// TIA Portal V17 export
// export: Created 2022-07-28T18:03:21.6529657Z, ExportSetting None, DisplayName Totally Integrated Automation Portal, DisplayVersion V17, DisplayName TIA Portal Openness, DisplayVersion V17, DisplayName TIA Portal Teamcenter Gateway, DisplayVersion V17, DisplayName TIA Portal Version Control Interface, DisplayVersion V17, DisplayName TIA Portal Test Suite Advanced, DisplayVersion V17, DisplayName SINAMICS Startdrive Advanced, DisplayVersion V17, DisplayName SINAMICS DCC, DisplayVersion V17, DisplayName SINAMICS Startdrive G130, G150, S120, S150, SINAMICS MV, S210, DisplayVersion V17, DisplayName SINAMICS Startdrive G110M, G120, G120C, G120D, G120P, G115D, DisplayVersion V17, DisplayName STEP 7 Professional, DisplayVersion V17, DisplayName SIMATIC Energy Suite, DisplayVersion V17, DisplayName STEP 7 CFC, DisplayVersion V17, DisplayName STEP 7 Safety, DisplayVersion V17, DisplayName WinCC Advanced / Unified PC, DisplayVersion V17, DisplayName SIMATIC Visualization Architect, DisplayVersion V17
TYPE "_SlideGate_Cond_StateBits"
   STRUCT
      Error { ExternalAccessible := 'False'; ExternalVisible := 'False'; ExternalWritable := 'False'} : Bool;   // x0 - 1 = [1-level alarm] -General alarm- Активна Загальна аварія(об'єднує усі аварії) / General alarm - Overall error
      Warning { ExternalAccessible := 'False'; ExternalVisible := 'False'; ExternalWritable := 'False'} : Bool;   // x1 - 1 = [2-level alarm] - Warning - Активне попередження (об'єднує усі попередження)
      Maintenance { ExternalAccessible := 'False'; ExternalVisible := 'False'; ExternalWritable := 'False'} : Bool;   // x2 - 1 = [3-level ] - Maintenance - Обслуговування - Спрацювали таймери/лічильники обслуговування
      Interlocked { ExternalAccessible := 'False'; ExternalVisible := 'False'; ExternalWritable := 'False'} : Bool;   // x3 - 1 = [Interlock] - Interloked - Заблоковано
      Ready { ExternalAccessible := 'False'; ExternalVisible := 'False'; ExternalWritable := 'False'} : Bool;   // x4 - 1 = Готовий - ...........
      Stoped { ExternalAccessible := 'False'; ExternalVisible := 'False'; ExternalWritable := 'False'} : Bool;   // x5 - 1 = Зупинений
      Run { ExternalAccessible := 'False'; ExternalVisible := 'False'; ExternalWritable := 'False'} : Bool;   // x6 - 1 = Запущено / напрямок руху Forward або Revers / Відкривається або Закривається
      RunOpen { ExternalAccessible := 'False'; ExternalVisible := 'False'; ExternalWritable := 'False'} : Bool;   // x7 - 1 = Запущено / напрямок руху Forward / Відкривається
      RunClose { ExternalAccessible := 'False'; ExternalVisible := 'False'; ExternalWritable := 'False'} : Bool;   // x8 - 1 = Запущено / напрямок руху Revers / Закривається
      bit_9 { ExternalAccessible := 'False'; ExternalVisible := 'False'; ExternalWritable := 'False'} : Bool;   // x9 -
      bit_10 { ExternalAccessible := 'False'; ExternalVisible := 'False'; ExternalWritable := 'False'} : Bool;   // x10 -
      Opened { ExternalAccessible := 'False'; ExternalVisible := 'False'; ExternalWritable := 'False'} : Bool;   // x11 - Повторює сигнал від кінцевика - відкрито
      Closed { ExternalAccessible := 'False'; ExternalVisible := 'False'; ExternalWritable := 'False'} : Bool;   // x12 - Повторює сигнал від кінцевика - закрито
      ActiveH { ExternalAccessible := 'False'; ExternalVisible := 'False'; ExternalWritable := 'False'} : Bool;   // x13 - 1 = HLevel is active
      ActiveL { ExternalAccessible := 'False'; ExternalVisible := 'False'; ExternalWritable := 'False'} : Bool;   // x14 - 1 = LLevel is active
      PumpIsAuto { ExternalAccessible := 'False'; ExternalVisible := 'False'; ExternalWritable := 'False'} : Bool;   // x15 - 1 = Choiced pump is in auto mode
      PumpIsReady { ExternalAccessible := 'False'; ExternalVisible := 'False'; ExternalWritable := 'False'} : Bool;   // x16 - 1 = Choiced pump is ready for start
      PumpIsRunning { ExternalAccessible := 'False'; ExternalVisible := 'False'; ExternalWritable := 'False'} : Bool;   // x17 - 1 = Choiced pump is running state
      bit_18 { ExternalAccessible := 'False'; ExternalVisible := 'False'; ExternalWritable := 'False'} : Bool;   // x18 - резер
      bit_19 { ExternalAccessible := 'False'; ExternalVisible := 'False'; ExternalWritable := 'False'} : Bool;   // x19 - резер
      bit_20 { ExternalAccessible := 'False'; ExternalVisible := 'False'; ExternalWritable := 'False'} : Bool;   // x20 - резер
      bit_21 { ExternalAccessible := 'False'; ExternalVisible := 'False'; ExternalWritable := 'False'} : Bool;   // x21 - резер
      Different { ExternalAccessible := 'False'; ExternalVisible := 'False'; ExternalWritable := 'False'} : Bool;   // x22 - (для групи) 1 = різні режими у об'єктів групи
      Disable { ExternalAccessible := 'False'; ExternalVisible := 'False'; ExternalWritable := 'False'} : Bool;   // x23 - 1 = Відключено/Виведено із експлуатації Function change to Stop mode
      ManualRemote { ExternalAccessible := 'False'; ExternalVisible := 'False'; ExternalWritable := 'False'} : Bool;   // x24 - 1 = Ручний дистанційний режим / керування із HMI / Manual Remote control mode
      Auto { ExternalAccessible := 'False'; ExternalVisible := 'False'; ExternalWritable := 'False'} : Bool;   // x25 - 1 = Автоматичний режим / Automatic mode Control - controlled via the CmdAuto...
      ManualLocal { ExternalAccessible := 'False'; ExternalVisible := 'False'; ExternalWritable := 'False'} : Bool;   // x26 - 1 = Ручний місцевий режим зі щита кнопками / Manual Local control mode
      Service { ExternalAccessible := 'False'; ExternalVisible := 'False'; ExternalWritable := 'False'} : Bool;   // x27 - 1 = Сервісний(+ManualRemote) ігноруються і не обробляються усі аварії/ блокування -Сontrol via HMI and no display of errors and warnings
      Repair { ExternalAccessible := 'False'; ExternalVisible := 'False'; ExternalWritable := 'False'} : Bool;   // x28 - 1 = Виведено на ремонт /функція не обробляється, аварії та блокування не виводяться, команди на фізичні виходи не передаються -No control is possible and no display of errors and warnings
      Independent { ExternalAccessible := 'False'; ExternalVisible := 'False'; ExternalWritable := 'False'} : Bool;   // x29 - 1 = Незалежний режим роботи - режими перемикаються як оператором так і командами CmdAuto/Global // 0 = режими перемикаються тільки командами CmdAuto/Global
      Simulation { ExternalAccessible := 'False'; ExternalVisible := 'False'; ExternalWritable := 'False'} : Bool;   // x30 - 1 = Симуляція - команди на фізичні виходи не передаються - входи/аварії/блокування можуть симулюватися або активовутися вручну
      "not used" { ExternalAccessible := 'False'; ExternalVisible := 'False'; ExternalWritable := 'False'} : Bool;   // x31 - not used
   END_STRUCT;
END_TYPE
